PROGRAM Axis_07_Function_Blocks
VAR
END_VAR

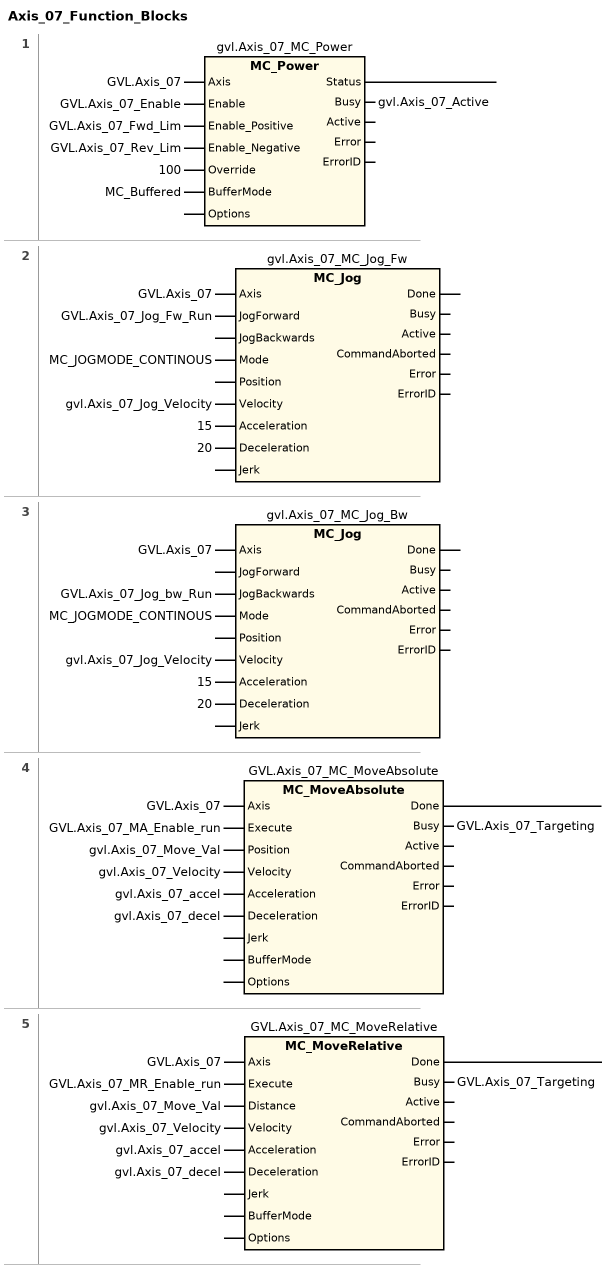
// NETWORK 1
gvl.Axis_07_MC_Power(
    Axis := GVL.Axis_07,
    Enable := GVL.Axis_07_Enable,
    Enable_Positive := GVL.Axis_07_Fwd_Lim,
    Enable_Negative := GVL.Axis_07_Rev_Lim,
    Override := 100,
    BufferMode := MC_Buffered,
    Busy => gvl.Axis_07_Active); // MC_Power

// NETWORK 2
gvl.Axis_07_MC_Jog_Fw(
    Axis := GVL.Axis_07,
    JogForward := GVL.Axis_07_Jog_Fw_Run,
    Mode := MC_JOGMODE_CONTINOUS,
    Velocity := gvl.Axis_07_Jog_Velocity,
    Acceleration := 15,
    Deceleration := 20); // MC_Jog

// NETWORK 3
gvl.Axis_07_MC_Jog_Bw(
    Axis := GVL.Axis_07,
    JogBackwards := GVL.Axis_07_Jog_bw_Run,
    Mode := MC_JOGMODE_CONTINOUS,
    Velocity := gvl.Axis_07_Jog_Velocity,
    Acceleration := 15,
    Deceleration := 20); // MC_Jog

// NETWORK 4
GVL.Axis_07_MC_MoveAbsolute(
    Axis := GVL.Axis_07,
    Execute := GVL.Axis_07_MA_Enable_run,
    Position := gvl.Axis_07_Move_Val,
    Velocity := gvl.Axis_07_Velocity,
    Acceleration := gvl.Axis_07_accel,
    Deceleration := gvl.Axis_07_decel,
    Busy => GVL.Axis_07_Targeting); // MC_MoveAbsolute

// NETWORK 5
GVL.Axis_07_MC_MoveRelative(
    Axis := GVL.Axis_07,
    Execute := GVL.Axis_07_MR_Enable_run,
    Distance := gvl.Axis_07_Move_Val,
    Velocity := gvl.Axis_07_Velocity,
    Acceleration := gvl.Axis_07_accel,
    Deceleration := gvl.Axis_07_decel,
    Busy => GVL.Axis_07_Targeting); // MC_MoveRelative

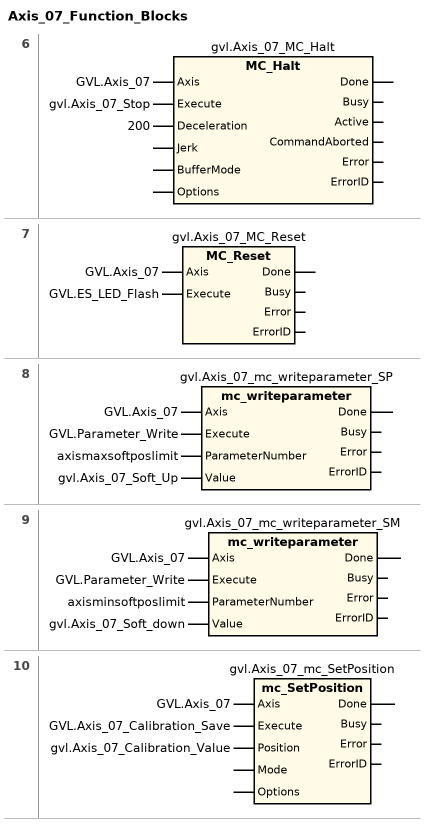
// NETWORK 6
gvl.Axis_07_MC_Halt(Axis := GVL.Axis_07, Execute := gvl.Axis_07_Stop, Deceleration := 200); // MC_Halt

// NETWORK 7
gvl.Axis_07_MC_Reset(Axis := GVL.Axis_07, Execute := GVL.ES_LED_Flash); // MC_Reset

// NETWORK 8
gvl.Axis_07_mc_writeparameter_SP(
    Axis := GVL.Axis_07,
    Execute := GVL.Parameter_Write,
    ParameterNumber := axismaxsoftposlimit,
    Value := gvl.Axis_07_Soft_Up); // mc_writeparameter

// NETWORK 9
gvl.Axis_07_mc_writeparameter_SM(
    Axis := GVL.Axis_07,
    Execute := GVL.Parameter_Write,
    ParameterNumber := axisminsoftposlimit,
    Value := gvl.Axis_07_Soft_down); // mc_writeparameter

// NETWORK 10
gvl.Axis_07_mc_SetPosition(
    Axis := GVL.Axis_07,
    Execute := GVL.Axis_07_Calibration_Save,
    Position := gvl.Axis_07_Calibration_Value); // mc_SetPosition

END_PROGRAM

(* stored: Version 1.1.0.1, ProductVersion 3.1.4022.12
   POU Axis_07_Function_Blocks: Id {55af5fd9-1245-416f-b69f-7c2d7cb08d17}, SpecialFunc None *)
